// TwinCAT 3 PLC project MAS418_PLC
// ProgramVersion: 3.1.4023.0
// libraries:
//   Tc2_Standard, * (Beckhoff Automation GmbH)
//   Tc2_System, * (Beckhoff Automation GmbH)
//   Tc3_Module, * (Beckhoff Automation GmbH)
//   VisuDialogs, * (System)
// project tree:
//   / GlobalTextList.TcGTLO, PlcTask.TcTTO, Visualization Manager.TcVMO (not stored)
//   POUs/ MAIN.TcPOU
//   VISUs/ HMI.TcVIS
// real-time tasks:
//   TASK PlcTask: cycle T#10ms, priority 20, ADS port 350

CONFIGURATION MAS418_PLC
    RESOURCE PLC ON TwinCAT3
        TASK PlcTask(INTERVAL := T#10ms, PRIORITY := 20);
        PROGRAM MAIN WITH PlcTask : MAIN;
    END_RESOURCE
END_CONFIGURATION

// ---- POUs/MAIN.TcPOU
PROGRAM MAIN

VAR
	bEnable : BOOL := FALSE;
	bStart : BOOL := FALSE;
	nINT : INT := -32768;
	nUNIT : UINT := 65535;
	fREAL : REAL := 255.255;
END_VAR

bEnable := bStart;

END_PROGRAM

// ---- GlobalTextList.TcGTLO
TEXTLIST GlobalTextList
  229 = '%f'
  218 = '%i'
  586 = 'DataTypeTesting'
  853 = 'GroupBox'
  924 = 'Power ON'
END_TEXTLIST

// ---- VISUs/HMI.TcVIS
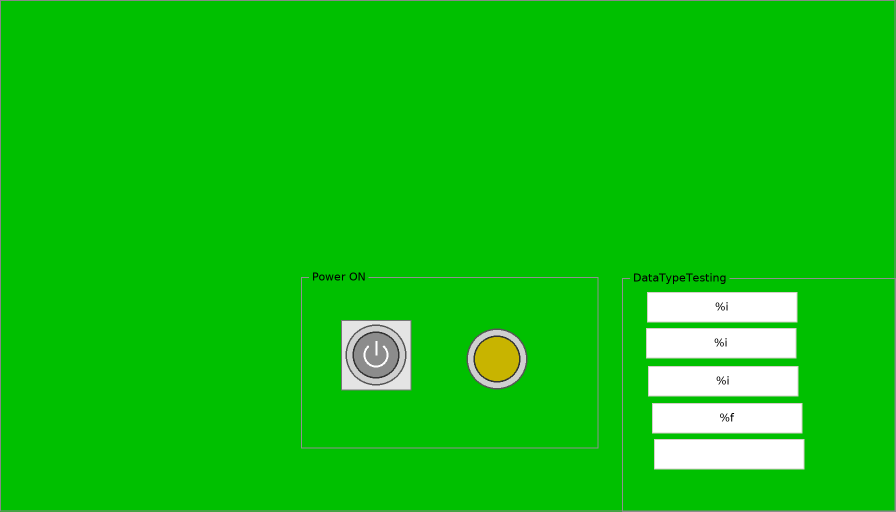
VISUALIZATION HMI  // 896x512
    GroupBox (301,269 297x179), "Power ON"
        PowerSwitch (40,51 70x70), variable: MAIN.bStart, behaviour: TOGGLE, style: Switch-PowerSwitch-Gray
        Lamp1 (161,55 70x70), variable: MAIN.bEnable, style: Lamp-Lamp1-Yellow
    GroupBox (622,270 274x242), "DataTypeTesting"
        Textfield (24,58 150x30), "%i", text variable: MAIN.nINT
        Textfield (26,96 150x30), "%i", text variable: MAIN.nUNIT
        Textfield (25,22 150x30), "%i", text variable: MAIN.bEnable
        Textfield (30,133 150x30), "%f", text variable: MAIN.fREAL
            OnMouseDown: write the text variable via Default
    Textfield (654,439 150x30)
END_VISUALIZATION
